FUNCTION MotorDegreeToCablePosition : LREAL
VAR_INPUT
	motor_position : LREAL;
END_VAR
VAR_OUTPUT
	cable_position : LREAL;
END_VAR
VAR
END_VAR

cable_position := motor_position;

END_FUNCTION

(* stored: Version 1.1.0.1, ProductVersion 3.1.4024.11
   POU MotorDegreeToCablePosition: Id {74506d61-801a-44fc-b9b8-372e062fd7c0}, SpecialFunc None *)
